(* IEC 61131-3 sources: Word/plc-course/12-data-structures/labs/solutions, 3 files *)

(* ---- 12-3-motor-array.st ---- *)
(* Lab 12-3: Four pumps, one data model, one loop.
   Module 12 (Data structures). REFERENCE SOLUTION - try the lab yourself first.

   Four identical feed pumps, P-101 to P-104. In CODESYS or TIA Portal you
   might declare ARRAY[1..4] OF FB_Motor and call each element in a loop.
   MATIEC (and so OpenPLC) has no arrays of function block instances and no
   FB instances inside a structure, so the design here keeps EVERYTHING a
   pump needs, including what a TON would have remembered, in a structure:

     ST_MotorData = Cmd (HMI -> PLC) + Cfg (settings) + Sts (PLC -> HMI)
                    + Alm (latched alarms) + the feedback and a timing counter

   and processes ARRAY[1..4] OF ST_MotorData with ONE function block instance
   that loops over the array once per scan. The timing is done with a
   millisecond clock: each pump counts the ms for which its command and its
   feedback have disagreed, instead of owning a TON.

   Training exercise: the area stop here is an ordinary control stop, not an
   emergency stop. Emergency stops belong in a safety system (Module 20). *)

TYPE
  E_MotorState : (Stopped, Starting, Running, Faulted);

  ST_MotorCmd :
  STRUCT                          (* HMI -> PLC. The HMI sets a bit; the PLC clears it. *)
    Start : BOOL;
    Stop  : BOOL;
    Reset : BOOL;                 (* clears latched alarms; never starts the pump *)
  END_STRUCT;

  ST_MotorCfg :
  STRUCT                          (* engineer settings (retentive and change-controlled on a real plant) *)
    FbTimeoutMs : DINT := 2000;   (* ms that command and feedback may disagree *)
  END_STRUCT;

  ST_MotorSts :
  STRUCT                          (* PLC -> HMI, written by the PLC every scan *)
    State  : E_MotorState;
    RunCmd : BOOL;                (* command to the contactor *)
    Starts : DINT;                (* successful starts (Starting -> Running) since power-up *)
  END_STRUCT;

  ST_MotorAlm :
  STRUCT                          (* PLC -> HMI, latched until Reset *)
    FailToStart : BOOL;           (* started, but no feedback within FbTimeoutMs *)
    FbLost      : BOOL;           (* was running, feedback gone for FbTimeoutMs *)
    Uncommanded : BOOL;           (* stopped, but feedback present for FbTimeoutMs *)
  END_STRUCT;

  ST_MotorData :
  STRUCT
    Cmd        : ST_MotorCmd;
    Cfg        : ST_MotorCfg;
    Sts        : ST_MotorSts;
    Alm        : ST_MotorAlm;
    RunFb      : BOOL;            (* run feedback, copied from the input by the mapping layer *)
    DisagreeMs : DINT;            (* internal: ms that RunCmd and RunFb have disagreed *)
  END_STRUCT;
END_TYPE

FUNCTION_BLOCK FB_MotorGroup
  (* Runs the motor logic for every element of Motors, once per call.
     Call it exactly once per scan. All per-pump memory is in the array
     elements; the only memory of its own is the clock value of the last call.

     Per pump:
       Stopped  --Start (no Stop, no StopAll)-->  Starting
       Starting --RunFb-->                        Running   (Starts + 1)
       Starting/Running --Stop or StopAll-->      Stopped
       any state but Faulted: command and feedback disagree for
         FbTimeoutMs --> Faulted, with the alarm that matches the state:
         Starting: FailToStart, Running: FbLost, Stopped: Uncommanded
       Faulted  --Reset-->                        Stopped   (never Starting)
     RunCmd is TRUE in Starting and Running only. Command bits are cleared
     after every call. *)
  VAR_IN_OUT
    Motors : ARRAY[1..4] OF ST_MotorData;
  END_VAR
  VAR_INPUT
    NowMs   : DINT;               (* free-running millisecond clock *)
    StopAll : BOOL;               (* TRUE = stop every pump (area stop) *)
  END_VAR
  VAR_OUTPUT
    RunningCount : INT;           (* pumps in state Running *)
    AnyFault     : BOOL;          (* at least one pump in state Faulted *)
  END_VAR
  VAR
    LastMs   : DINT;              (* NowMs at the previous call *)
    ScanMs   : DINT;              (* ms since the previous call *)
    i        : INT;
    Disagree : BOOL;
  END_VAR
  VAR CONSTANT
    NO_CMD    : ST_MotorCmd := (Start := FALSE, Stop := FALSE, Reset := FALSE);
    NO_ALARMS : ST_MotorAlm := (FailToStart := FALSE, FbLost := FALSE, Uncommanded := FALSE);
  END_VAR

  ScanMs := NowMs - LastMs;
  LastMs := NowMs;
  RunningCount := 0;
  AnyFault := FALSE;

  FOR i := 1 TO 4 DO
    (* -- Reset clears the alarms and leaves a faulted pump stopped. If the
       cause is still there, the alarm comes back after another full
       FbTimeoutMs. The timing restarts only for a FAULTED pump: a Reset
       pressed while a disagreement is still being timed must not postpone
       (and so hide) the alarm. -- *)
    IF Motors[i].Cmd.Reset THEN
      Motors[i].Alm := NO_ALARMS;
      IF Motors[i].Sts.State = E_MotorState#Faulted THEN
        Motors[i].Sts.State := E_MotorState#Stopped;
        Motors[i].DisagreeMs := 0;
      END_IF;
    END_IF;

    (* -- Commands. Stop (and the area stop) win over Start. A start is only
       accepted from Stopped, so a faulted pump cannot be started. -- *)
    CASE Motors[i].Sts.State OF
      E_MotorState#Stopped:
        IF Motors[i].Cmd.Start AND NOT Motors[i].Cmd.Stop AND NOT StopAll THEN
          Motors[i].Sts.State := E_MotorState#Starting;
        END_IF;
      E_MotorState#Starting, E_MotorState#Running:
        IF Motors[i].Cmd.Stop OR StopAll THEN
          Motors[i].Sts.State := E_MotorState#Stopped;
        END_IF;
    END_CASE;

    (* -- Feedback proves the start. -- *)
    IF Motors[i].Sts.State = E_MotorState#Starting AND Motors[i].RunFb THEN
      Motors[i].Sts.State := E_MotorState#Running;
      Motors[i].Sts.Starts := Motors[i].Sts.Starts + 1;
    END_IF;

    (* -- Supervision: this pump's "timer" is a counter of milliseconds in the
       structure. It restarts whenever command and feedback agree, and it
       stops counting at the timeout (like a TON's ET stops at PT), so it
       cannot overflow however long a disagreement lasts. -- *)
    Motors[i].Sts.RunCmd := Motors[i].Sts.State = E_MotorState#Starting
                            OR Motors[i].Sts.State = E_MotorState#Running;
    Disagree := Motors[i].Sts.RunCmd XOR Motors[i].RunFb;
    IF NOT Disagree THEN
      Motors[i].DisagreeMs := 0;
    ELSIF Motors[i].DisagreeMs < Motors[i].Cfg.FbTimeoutMs THEN
      Motors[i].DisagreeMs := Motors[i].DisagreeMs + ScanMs;
    END_IF;

    IF Motors[i].DisagreeMs >= Motors[i].Cfg.FbTimeoutMs THEN
      CASE Motors[i].Sts.State OF
        E_MotorState#Starting: Motors[i].Alm.FailToStart := TRUE;
        E_MotorState#Running:  Motors[i].Alm.FbLost := TRUE;
        E_MotorState#Stopped:  Motors[i].Alm.Uncommanded := TRUE;
      END_CASE;
      Motors[i].Sts.State := E_MotorState#Faulted;
    END_IF;

    (* -- Final command and the group summary. -- *)
    Motors[i].Sts.RunCmd := Motors[i].Sts.State = E_MotorState#Starting
                            OR Motors[i].Sts.State = E_MotorState#Running;
    IF Motors[i].Sts.State = E_MotorState#Running THEN
      RunningCount := RunningCount + 1;
    END_IF;
    IF Motors[i].Sts.State = E_MotorState#Faulted THEN
      AnyFault := TRUE;
    END_IF;

    Motors[i].Cmd := NO_CMD;              (* every command bit is acted on once *)
  END_FOR;
END_FUNCTION_BLOCK

PROGRAM FeedPumps
  VAR (* physical inputs *)
    P101_RunFb AT %IX0.0 : BOOL;          (* P-101 contactor auxiliary contact *)
    P102_RunFb AT %IX0.1 : BOOL;          (* P-102 contactor auxiliary contact *)
    P103_RunFb AT %IX0.2 : BOOL;          (* P-103 contactor auxiliary contact *)
    P104_RunFb AT %IX0.3 : BOOL;          (* P-104 discharge flow switch (slow to make) *)
    StopAll_NC AT %IX1.0 : BOOL;          (* area stop push-button, NC: TRUE = healthy *)
  END_VAR
  VAR (* physical outputs *)
    P101_Contactor AT %QX0.0 : BOOL;
    P102_Contactor AT %QX0.1 : BOOL;
    P103_Contactor AT %QX0.2 : BOOL;
    P104_Contactor AT %QX0.3 : BOOL;
    FaultLamp      AT %QX0.4 : BOOL;      (* ON while any pump is faulted *)
  END_VAR
  VAR (* the data model: one element per pump, read and written by the HMI.
         Cfg.FbTimeoutMs starts at the ST_MotorCfg default of 2000 ms; the
         first-scan block gives P-104 its 5000 ms. *)
    Motors : ARRAY[1..4] OF ST_MotorData;
    RunningCount : INT;                   (* pumps proven running *)
  END_VAR
  VAR (* clock - given, do not change *)
    UpTime : TON;
    NowMs  : DINT;                        (* ms since power-up *)
  END_VAR
  VAR
    Initialised : BOOL;                   (* NOT retentive: FALSE until the first-scan block has run *)
    Group : FB_MotorGroup;                (* ONE instance for all four pumps *)
  END_VAR

  (* ---- First scan only (given): P-104's flow switch is slow to make, so it
     gets 5000 ms instead of the default 2000 ms. Standard IEC 61131-3 would
     say this in the declaration, with an initialiser for the array of
     structures:
       Motors : ARRAY[1..4] OF ST_MotorData := [3((Cfg := (FbTimeoutMs := 2000))),
                                                 (Cfg := (FbTimeoutMs := 5000))];
     OpenPLC's compiler does not accept this initialiser (see Appendix E), so
     the value is set here, at the very top, before the pump logic first
     reads it. Pumps 1 to 3 keep the default from ST_MotorCfg. Initialised
     is not RETAIN, so every restart starts again from these values, as the
     initialiser would. (Cfg is retentive on a real plant; Initialised would
     then have to be RETAIN too, or a warm restart would undo the engineer's
     settings.) ---- *)
  IF NOT Initialised THEN
    Motors[4].Cfg.FbTimeoutMs := 5000;
    Initialised := TRUE;
  END_IF;

  (* ---- Millisecond clock (given): see Lab 12-2. ---- *)
  UpTime(IN := TRUE, PT := T#24d);
  NowMs := LREAL_TO_DINT(TIME_TO_LREAL(UpTime.ET) / TIME_TO_LREAL(T#1s) * 1000.0);

  (* ---- Input mapping. Located variables cannot be arrays in MATIEC, so
     each input is copied into its element by hand, here and only here. ---- *)
  Motors[1].RunFb := P101_RunFb;
  Motors[2].RunFb := P102_RunFb;
  Motors[3].RunFb := P103_RunFb;
  Motors[4].RunFb := P104_RunFb;

  (* ---- All four pumps, one call. ---- *)
  Group(Motors := Motors, NowMs := NowMs, StopAll := NOT StopAll_NC);
  RunningCount := Group.RunningCount;

  (* ---- Output mapping: the one place each output is written. ---- *)
  P101_Contactor := Motors[1].Sts.RunCmd;
  P102_Contactor := Motors[2].Sts.RunCmd;
  P103_Contactor := Motors[3].Sts.RunCmd;
  P104_Contactor := Motors[4].Sts.RunCmd;
  FaultLamp := Group.AnyFault;
END_PROGRAM

CONFIGURATION Config0
  RESOURCE Res0 ON PLC
    TASK MainTask(INTERVAL := T#10ms, PRIORITY := 0);
    PROGRAM Inst0 WITH MainTask : FeedPumps;
  END_RESOURCE
END_CONFIGURATION

(* ---- 12-1-recipe-manager.st ---- *)
(* Lab 12-1: Recipe manager - an array of structures, validated before use.
   Module 12 (Data structures). REFERENCE SOLUTION - try the lab yourself first.

   A jacketed mixing vessel makes five products. Each product's recipe is a
   structure (name, three ingredient doses, temperature, mixing time), and the
   recipe book is an ARRAY[1..5] OF ST_Recipe that the operator edits on the
   HMI. The batch sequence never uses the book directly: it uses Active, a
   validated copy taken when the operator presses Load.

   Design points shown here:
   - the index from the HMI is checked BEFORE Recipes[SelectNo] is touched;
   - the value checks live in a FUNCTION that takes the recipe and the limits
     as structures, so the same check serves the live "Load" button status and
     the load itself;
   - the load is all-or-nothing: one whole-structure assignment, only after
     every check has passed. A rejected load leaves Active exactly as it was. *)

TYPE
  ST_Recipe :
  STRUCT
    Name    : STRING;               (* product name shown on the HMI; '' = empty slot *)
    Dose    : ARRAY[1..3] OF REAL;  (* kg of ingredient 1 (water), 2 (base), 3 (seasoning) *)
    Temp    : REAL;                 (* degC, batch temperature setpoint *)
    MixTime : TIME;                 (* mixing time once the batch is at temperature *)
  END_STRUCT;

  ST_RecipeLimits :
  STRUCT
    DoseMax    : REAL;              (* kg, largest dose of any one ingredient *)
    TotalMax   : REAL;              (* kg, vessel working capacity *)
    TempMin    : REAL;              (* degC *)
    TempMax    : REAL;              (* degC *)
    MixTimeMin : TIME;
    MixTimeMax : TIME;
  END_STRUCT;

  (* Result of the last load command. The first value is the initial value. *)
  E_LoadResult : (NotLoaded, Loaded, BadIndex, EmptySlot, BadValue, BatchBusy);
END_TYPE

FUNCTION F_RecipeValuesOk : BOOL
  (* TRUE when every number in the recipe is inside its limits (all limits
     inclusive). The name is the caller's business. Guard-clause style: the
     result starts FALSE and each failed check leaves at once with RETURN. *)
  VAR_INPUT
    R   : ST_Recipe;          (* the recipe to check (passed by value: a copy) *)
    Lim : ST_RecipeLimits;    (* the limits, also a structure *)
  END_VAR
  VAR
    i     : INT;
    Total : REAL;             (* kg, sum of the three doses *)
  END_VAR

  F_RecipeValuesOk := FALSE;              (* guilty until proven innocent *)

  Total := 0.0;
  FOR i := 1 TO 3 DO
    IF R.Dose[i] < 0.0 OR R.Dose[i] > Lim.DoseMax THEN
      RETURN;                             (* one bad dose rejects the recipe *)
    END_IF;
    Total := Total + R.Dose[i];
  END_FOR;

  (* A cross-check that no single field can make: three legal doses can
     still overfill the vessel. An all-zero recipe is meaningless too. *)
  IF Total <= 0.0 OR Total > Lim.TotalMax THEN
    RETURN;
  END_IF;

  IF R.Temp < Lim.TempMin OR R.Temp > Lim.TempMax THEN
    RETURN;
  END_IF;

  IF R.MixTime < Lim.MixTimeMin OR R.MixTime > Lim.MixTimeMax THEN
    RETURN;
  END_IF;

  F_RecipeValuesOk := TRUE;
END_FUNCTION

PROGRAM RecipeManager
  VAR (* recipe book, edited on the HMI recipe screen. Slots 1 to 4 are
         filled in by the first-scan block at the top of the code. Slot 4
         holds a typing mistake (95 degC), and slot 5 is left empty on
         purpose ('', 0.0 and T#0s). Both must be refused. *)
    Recipes : ARRAY[1..5] OF ST_Recipe;
  END_VAR
  VAR (* HMI selection and command, and the state of the batch *)
    SelectNo     : INT;             (* recipe number chosen on the HMI; 0 = none *)
    LoadCmd      : BOOL;            (* HMI sets it to request a load; the PLC clears it *)
    BatchRunning : BOOL;            (* TRUE while a batch is in progress (from the sequence) *)
  END_VAR
  VAR (* results - keep these names *)
    SelectedOk   : BOOL;            (* the selected recipe could be loaded (enables the Load button) *)
    Active       : ST_Recipe;       (* the recipe the batch sequence uses *)
    ActiveNo     : INT;             (* which slot Active came from; 0 = nothing loaded yet *)
    LoadResult   : E_LoadResult;    (* outcome of the last load command *)
  END_VAR
  VAR (* the limits of this vessel: set by the first-scan block, never written anywhere else *)
    RecipeLimits : ST_RecipeLimits;
  END_VAR
  VAR CONSTANT
    FIRST_SLOT : INT := 1;          (* keep in step with the ARRAY[1..5] bounds *)
    LAST_SLOT  : INT := 5;
  END_VAR
  VAR
    Initialised : BOOL;             (* NOT retentive: FALSE until the first-scan block has run *)
    Check : E_LoadResult;           (* what a load of the selected slot would give now *)
  END_VAR

  (* ---- 0. First scan only: fill in the recipe book and the limits.
     Standard IEC 61131-3 would give both as initialisers in the declarations:
       Recipes : ARRAY[1..5] OF ST_Recipe := [
         (Name := 'Tomato soup', Dose := [400.0, 150.0, 20.0], Temp := 85.0, MixTime := T#20m),
         ...];
       RECIPE_LIMITS : ST_RecipeLimits := (DoseMax := 500.0, ...);   (a VAR CONSTANT)
     OpenPLC's compiler does not accept these initialisers (see Appendix E),
     so the values are set here. The block is at the very top, so the values
     are in place before anything below reads them, from the first scan on.
     Initialised is not RETAIN, so every restart starts again from these
     values, as the initialisers would. (If the book were RETAIN, as it would
     be on a real plant, Initialised would have to be RETAIN too, or every
     warm restart would overwrite the operator's edits.) ---- *)
  IF NOT Initialised THEN
    Recipes[1].Name := 'Tomato soup';
    Recipes[1].Dose[1] := 400.0;  Recipes[1].Dose[2] := 150.0;  Recipes[1].Dose[3] := 20.0;
    Recipes[1].Temp := 85.0;      Recipes[1].MixTime := T#20m;

    Recipes[2].Name := 'Vegetable stock';
    Recipes[2].Dose[1] := 450.0;  Recipes[2].Dose[2] := 300.0;  Recipes[2].Dose[3] := 10.0;
    Recipes[2].Temp := 80.0;      Recipes[2].MixTime := T#30m;

    Recipes[3].Name := 'Cheese sauce';
    Recipes[3].Dose[1] := 250.0;  Recipes[3].Dose[2] := 200.0;  Recipes[3].Dose[3] := 50.0;
    Recipes[3].Temp := 65.0;      Recipes[3].MixTime := T#15m;

    Recipes[4].Name := 'Trial batch';
    Recipes[4].Dose[1] := 100.0;  Recipes[4].Dose[2] := 100.0;  Recipes[4].Dose[3] := 0.0;
    Recipes[4].Temp := 95.0;      Recipes[4].MixTime := T#10m;   (* 95 degC: the typing mistake *)

    (* slot 5 is left empty *)

    RecipeLimits.DoseMax    := 500.0;     (* kg, largest dose of any one ingredient *)
    RecipeLimits.TotalMax   := 1000.0;    (* kg, vessel working capacity *)
    RecipeLimits.TempMin    := 20.0;      (* degC *)
    RecipeLimits.TempMax    := 85.0;      (* degC *)
    RecipeLimits.MixTimeMin := T#1m;
    RecipeLimits.MixTimeMax := T#2h;

    Initialised := TRUE;
  END_IF;

  (* ---- 1. Check the selected slot, every scan. The index comes from the
     HMI, so it is tested FIRST: Recipes[SelectNo] is only read inside the
     ELSIF branches, which run only when the index is in range. ---- *)
  IF SelectNo < FIRST_SLOT OR SelectNo > LAST_SLOT THEN
    Check := E_LoadResult#BadIndex;
  ELSIF LEN(Recipes[SelectNo].Name) = 0 THEN
    Check := E_LoadResult#EmptySlot;
  ELSIF NOT F_RecipeValuesOk(R := Recipes[SelectNo], Lim := RecipeLimits) THEN
    Check := E_LoadResult#BadValue;
  ELSE
    Check := E_LoadResult#Loaded;   (* passes every check: it can be loaded *)
  END_IF;

  SelectedOk := Check = E_LoadResult#Loaded;

  (* ---- 2. The load command: acted on once, then cleared (the HMI sets
     command bits, the PLC clears them). Never change the recipe of a batch
     that is running. ---- *)
  IF LoadCmd THEN
    IF BatchRunning THEN
      LoadResult := E_LoadResult#BatchBusy;
    ELSE
      LoadResult := Check;
      IF Check = E_LoadResult#Loaded THEN
        Active := Recipes[SelectNo];      (* whole-structure copy: all or nothing *)
        ActiveNo := SelectNo;
      END_IF;
    END_IF;
    LoadCmd := FALSE;
  END_IF;
END_PROGRAM

CONFIGURATION Config0
  RESOURCE Res0 ON PLC
    TASK MainTask(INTERVAL := T#10ms, PRIORITY := 0);
    PROGRAM Inst0 WITH MainTask : RecipeManager;
  END_RESOURCE
END_CONFIGURATION

(* ---- 12-2-event-log.st ---- *)
(* Lab 12-2: Event log - a ring buffer of structures.
   Module 12 (Data structures). REFERENCE SOLUTION - try the lab yourself first.

   A pump station keeps its last ten events (trips, alarms, operator actions)
   in the PLC, so that the HMI can show them and a historian can collect them.
   Each event is a structure: a code and a time stamp in milliseconds.

   The log is a RING BUFFER: entries are written into ten fixed slots,
   EventLog[0], [1], ... [9], then [0] again, and only the index Newest moves.
   Nothing is ever shifted, so logging costs the same however full the log
   is, and a reader always finds an entry in the slot where it was written.
   When the log is full, each new event overwrites the oldest one.

   Arithmetic used: next slot = (Newest + 1) MOD 10, and the slot of the event
   "Age" events back = (Newest - Age + 10) MOD 10. The "+ 10" matters: MOD
   keeps the sign of the dividend, so (0 - 1) MOD 10 is -1, not 9. *)

TYPE
  ST_Event :
  STRUCT
    Code  : INT;    (* event code, 1..32767; 0 = empty entry *)
    Stamp : DINT;   (* ms since power-up when the event was logged *)
  END_STRUCT;
END_TYPE

PROGRAM EventLogger
  VAR (* requests from the rest of the program and the HMI *)
    NewCode  : INT;                      (* code of the event to log *)
    LogReq   : BOOL;                     (* TRUE = log NewCode now; the logger clears it *)
    ClearCmd : BOOL;                     (* TRUE = empty the log; the logger clears it *)
    ViewAge  : INT;                      (* HMI: 0 = newest event, 1 = the one before, ... *)
  END_VAR
  VAR (* the log - keep these names *)
    EventLog : ARRAY[0..9] OF ST_Event;  (* the ring: ten fixed slots *)
    Newest   : INT;                      (* slot of the newest entry (0 while the log is empty) *)
    Count    : INT;                      (* valid entries, 0..10 *)
    Total    : DINT;                     (* events logged since power-up or the last clear *)
    View     : ST_Event;                 (* the event ViewAge events back from the newest *)
    ViewValid : BOOL;                    (* TRUE when View holds a real event *)
  END_VAR
  VAR (* clock - given, do not change *)
    UpTime   : TON;
    NowMs    : DINT;                     (* ms since power-up *)
  END_VAR
  VAR CONSTANT
    LOG_SIZE : INT := 10;                (* keep in step with ARRAY[0..9] *)
    NO_EVENT : ST_Event := (Code := 0, Stamp := 0);
  END_VAR
  VAR
    i        : INT;
    ViewSlot : INT;
  END_VAR

  (* ---- 0. Millisecond clock (given). TIME_TO_LREAL gives seconds in
     MATIEC and milliseconds in CODESYS; dividing by TIME_TO_LREAL(T#1s)
     gives seconds on both, and * 1000.0 makes milliseconds. The TON's ET
     stops at PT, so this clock is good for 24 days: fine for a lab. ---- *)
  UpTime(IN := TRUE, PT := T#24d);
  NowMs := LREAL_TO_DINT(TIME_TO_LREAL(UpTime.ET) / TIME_TO_LREAL(T#1s) * 1000.0);

  (* ---- 1. Clear: empty every slot and start again at slot 0. ---- *)
  IF ClearCmd THEN
    FOR i := 0 TO LOG_SIZE - 1 DO
      EventLog[i] := NO_EVENT;           (* whole-structure assignment *)
    END_FOR;
    Newest := 0;
    Count := 0;
    Total := 0;
    ClearCmd := FALSE;
  END_IF;

  (* ---- 2. Log one event per request. Codes 0 and below are not events:
     the request is dropped (and still cleared). ---- *)
  IF LogReq THEN
    IF NewCode > 0 THEN
      IF Count > 0 THEN
        Newest := (Newest + 1) MOD LOG_SIZE;   (* step on, wrapping 9 -> 0 *)
      END_IF;                                  (* the first entry goes into slot 0 *)
      EventLog[Newest].Code := NewCode;
      EventLog[Newest].Stamp := NowMs;
      IF Count < LOG_SIZE THEN
        Count := Count + 1;                    (* once full, Count stays 10 and the
                                                  oldest entry has just been overwritten *)
      END_IF;
      Total := Total + 1;
    END_IF;
    LogReq := FALSE;
  END_IF;

  (* ---- 3. View for the HMI, every scan. ViewAge comes from the HMI, so it
     is checked against Count before it is used to find a slot. ---- *)
  IF ViewAge >= 0 AND ViewAge < Count THEN
    ViewSlot := (Newest - ViewAge + LOG_SIZE) MOD LOG_SIZE;
    View := EventLog[ViewSlot];
    ViewValid := TRUE;
  ELSE
    View := NO_EVENT;
    ViewValid := FALSE;
  END_IF;
END_PROGRAM

CONFIGURATION Config0
  RESOURCE Res0 ON PLC
    TASK MainTask(INTERVAL := T#10ms, PRIORITY := 0);
    PROGRAM Inst0 WITH MainTask : EventLogger;
  END_RESOURCE
END_CONFIGURATION
